FUNCTION_BLOCK PuestoManual
VAR_INPUT
	SFCreset:BOOL;
	Reset:BOOL;
	Enable:BOOL;
	FinCiclo:BOOL;
	SensorPallet:BOOL;
	Pulsador1 AT %I*:BOOL;
	NumeroDePuesto :INT;
	
END_VAR
VAR_OUTPUT
	StopperOFF AT %Q*:BOOL;
	Centrador AT%Q*:BOOL;
	LuzRoja AT%Q*:BOOL;
	FinPuesto:BOOL;
	SalidaAlarma:BOOL;
	EnMovimiento:BOOL;
	EsperandoPalet :BOOL;
	RetrasoPuesto :INT;
END_VAR
VAR
END_VAR

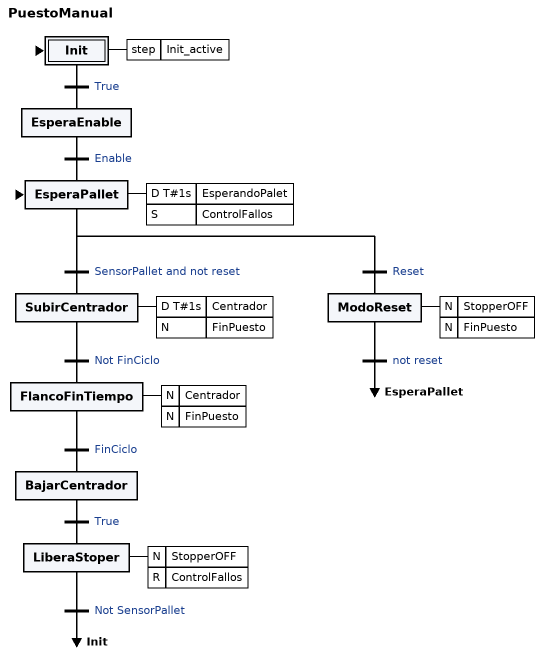
INITIAL_STEP Init:
    Init_active(N);  // step action
END_STEP
TRANSITION FROM Init TO EsperaEnable
    := True;
END_TRANSITION
STEP EsperaEnable:
END_STEP
TRANSITION FROM EsperaEnable TO EsperaPallet
    := Enable;
END_TRANSITION
STEP EsperaPallet:
    EsperandoPalet(D, T#1s);
    ControlFallos(S);
END_STEP
TRANSITION FROM EsperaPallet TO SubirCentrador
    := SensorPallet and not reset;
END_TRANSITION
STEP SubirCentrador:  // min time T#1s
    Centrador(D, T#1s);
    FinPuesto(N);
END_STEP
TRANSITION FROM SubirCentrador TO FlancoFinTiempo
    := Not FinCiclo;
END_TRANSITION
STEP FlancoFinTiempo:
    Centrador(N);
    FinPuesto(N);
END_STEP
TRANSITION FROM FlancoFinTiempo TO BajarCentrador
    := FinCiclo;
END_TRANSITION
STEP BajarCentrador:  // min time T#1s
END_STEP
TRANSITION FROM BajarCentrador TO LiberaStoper
    := True;
END_TRANSITION
TRANSITION FROM EsperaPallet TO ModoReset
    := Reset;
END_TRANSITION
STEP ModoReset:
    StopperOFF(N);
    FinPuesto(N);
END_STEP
TRANSITION FROM ModoReset TO EsperaPallet
    := not reset;
END_TRANSITION
STEP LiberaStoper:  // min time T#1s
    StopperOFF(N);
    ControlFallos(R);
END_STEP
TRANSITION FROM LiberaStoper TO Init
    := Not SensorPallet;
END_TRANSITION

ACTION ControlFallos:

IF GVL.FalloPallet[NumeroDePuesto] THEN
	LuzRoja :=TRUE;
	FinPuesto := FALSE;
ELSE
	LuzRoja :=FALSE;
	FinPuesto := TRUE;
END_IF


IF GVL.FalloPallet[NumeroDePuesto] AND Pulsador1 THEN
	GVL.FalloPallet[NumeroDePuesto] := FALSE;
END_IF
END_ACTION

ACTION Init_active:
LuzRoja := FALSE;
FinPUesto :=FALSE;
SFCreset:=FALSE;
END_ACTION

END_FUNCTION_BLOCK

(* stored: Version 1.1.0.1, ProductVersion 3.1.4024.3
   POU PuestoManual: Id {21341ffa-e029-442c-ab2b-4a959c0a407a}, SpecialFunc None
   Action ControlFallos: Id {577e7555-a673-4f73-b028-be1352e85e1d}
   Action Init_active: Id {14025df9-9ec7-494b-b463-d846ee8ef1de} *)
